# EPICS substitutions: src/makeBaseApp/top/pcdsModuleLib/Db/_APPNAME_.substitutions
#
# _APPNAME_ database substitutions file
#

# Generate _APPNAME_ db file
#	Macros:
#		TODO:	List here any macros used in the template
#				Note which ones have defaults.
file __APPNAME_.template
{
	{
		# Hack till msi supports empty substitutions
		IOC		=	$(IOC),
	}
}
